// Mitsubishi GX Works2 project: KhanhHungTap2FX3U   PLC: FX3U/FX3UC

// global labels: Global1
VAR_GLOBAL
  XXLimitN AT M8344 : BOOL;
  XXLimitP AT M8343 : BOOL;
  XXBusy AT M8340 : BOOL;
  XXInterruptInverse AT M8347 : BOOL;
  XXPos AT D8340 : DINT;
  XXAccelTime AT D8348 : INT;
  XXDecelTime AT D8349 : INT;
  XXPosView AT D0 : DINT;
  XXTarPos AT D2 : DINT;
  XXFeed AT D4 : DINT;
  XXPPR AT D6 : DINT;
  XXTarR AT M0 : BOOL;
  XXTarRSkip AT D8 : INT;
  XXOn AT M1 : BOOL;
  XXRun AT M2 : BOOL;
  XXDirection AT M3 : BOOL;
  XXMinI AT X000 : BOOL;
  XXReadyI AT X004 : BOOL;
  XXPulseO AT Y000 : BOOL;
  XXDirectionO AT Y004 : BOOL;
  XXOnO AT Y003 : BOOL;
  YYLimitN AT M8354 : BOOL;
  YYLimitP AT M8353 : BOOL;
  YYBusy AT M8350 : BOOL;
  YYInterruptInverse AT M8357 : BOOL;
  YYPos AT D8350 : DINT;
  YYAccelTime AT D8358 : INT;
  YYDecelTime AT D8359 : INT;
  YYPosView AT D9 : DINT;
  YYTarPos AT D11 : DINT;
  YYFeed AT D13 : DINT;
  YYPPM AT D15 : DINT;
  YYTarR AT M4 : BOOL;
  YYTarRSkip AT D17 : INT;
  YYOn AT M5 : BOOL;
  YYRun AT M6 : BOOL;
  YYDirection AT M7 : BOOL;
  YYMinI AT X001 : BOOL;
  YYReadyI AT X005 : BOOL;
  YYPulseO AT Y001 : BOOL;
  YYDirectionO AT Y005 : BOOL;
  YYOnO AT Y007 : BOOL;
  ZZLimitN AT M8364 : BOOL;
  ZZLimitP AT M8363 : BOOL;
  ZZBusy AT M8360 : BOOL;
  ZZInterruptInverse AT M8367 : BOOL;
  ZZPos AT D8360 : DINT;
  ZZAccelTime AT D8368 : INT;
  ZZDecelTime AT D8369 : INT;
  ZZPosView AT D18 : DINT;
  ZZTarPos AT D20 : DINT;
  ZZFeed AT D22 : DINT;
  ZZPPR AT D24 : DINT;
  ZZTarR AT M8 : BOOL;
  ZZTarRSkip AT D26 : INT;
  ZZRun AT M9 : BOOL;
  ZZDirection AT M10 : BOOL;
  ZZReadyI AT X006 : BOOL;
  ZZPulseO AT Y002 : BOOL;
  ZZDirectionO AT Y006 : BOOL;
  ZZOnO AT Y010 : BOOL;
  Run AT M11 : BOOL;
  RunI AT X002 : BOOL;
  RunStop AT M12 : BOOL;
  RunStopI AT X003 : BOOL;
  RunState AT D27 : INT;
  RunStateNext AT M13 : BOOL;
  AxisSpinState AT D28 : INT;
  AxisSpinStateNext AT M14 : BOOL;
  AxisTapState AT D29 : INT;
  AxisTapStateNext AT M15 : BOOL;
  FoilExtractState AT D30 : INT;
  FoilExtractStateNext AT M16 : BOOL;
  FoilClampState AT D31 : INT;
  FoilClampStateNext AT M17 : BOOL;
  FoilSupplyState AT D32 : INT;
  FoilSupplyStateNext AT M18 : BOOL;
  FoilExtractDropN AT M19 : BOOL;
  FoilExtractDropNTimer AT TC0 : BOOL;
  FoilExtractDropNTimerDelay AT D33 : INT;
  FoilExtractDropP AT M20 : BOOL;
  FoilExtractDropPTimer AT TC1 : BOOL;
  FoilExtractDropPTimerDelay AT D34 : INT;
  FoilExtractDrop AT M21 : BOOL;
  FoilExtractDropO AT Y011 : BOOL;
  FoilExtractPushN AT M22 : BOOL;
  FoilExtractPushNTimer AT TC2 : BOOL;
  FoilExtractPushNTimerDelay AT D35 : INT;
  FoilExtractPushP AT M23 : BOOL;
  FoilExtractPushPTimer AT TC3 : BOOL;
  FoilExtractPushPTimerDelay AT D36 : INT;
  FoilExtractPush AT M24 : BOOL;
  FoilExtractPushO AT Y012 : BOOL;
  FoilClampN AT M25 : BOOL;
  FoilClampNTimer AT TC4 : BOOL;
  FoilClampNTimerDelay AT D37 : INT;
  FoilClampP AT M26 : BOOL;
  FoilClampPTimer AT TC5 : BOOL;
  FoilClampPTimerDelay AT D38 : INT;
  FoilClampNI AT X007 : BOOL;
  FoilClampPI AT X010 : BOOL;
  FoilClamp AT M27 : BOOL;
  FoilClampO AT Y013 : BOOL;
  FoilSupplyN AT M28 : BOOL;
  FoilSupplyNTimer AT TC6 : BOOL;
  FoilSupplyNTimerDelay AT D39 : INT;
  FoilSupplyP AT M29 : BOOL;
  FoilSupplyPTimer AT TC7 : BOOL;
  FoilSupplyPTimerDelay AT D40 : INT;
  FoilSupply AT M30 : BOOL;
  FoilSupplyO AT Y014 : BOOL;
  WorkFeedSpin AT D41 : DINT;
  WorkFeedTapSpin AT D43 : DINT;
  WorkFeedTapSpinUp AT D45 : DINT;
  FoilFull AT M31 : BOOL;
  FoilFullI AT X011 : BOOL;
  FoilFullTimer AT TC8 : BOOL;
  SpinArray AT D47 : ARRAY [0..7] OF DINT;
  SpinArrayIndex AT D63 : INT;
  SpinTest AT M32 : BOOL;
  SpinTestTimer AT TC9 : BOOL;
  SpinTestTimerDelay AT D64 : INT;
  SettingTapPitchI AT X012 : BOOL;
  SettingTapPitch AT D65 : DINT;
  SettingTapSpinSpeed1I AT X013 : BOOL;
  SettingTapSpinSpeed2I AT X014 : BOOL;
  SettingTapTravelBegin AT D67 : DINT;
  SettingFoilSupplyI AT X015 : BOOL;
  AirReady AT M33 : BOOL;
  AirReadyI AT X016 : BOOL;
  TapMoveToTravelBegin AT M34 : BOOL;
  TapCount AT D69 : DINT;
  TapCountAtSupplyEnd AT D71 : DINT;
  StopTap AT M35 : BOOL;
  StopTapTimer AT TC10 : BOOL;
  StopClamp AT M36 : BOOL;
  StopClampPLS AT M37 : BOOL;
  StopClampTimer AT TC11 : BOOL;
  FoilSupplyPTimeoutTimer AT TC12 : BOOL;
  FoilSupplyPTimeoutTimerDelay AT D73 : INT;
  XXOff AT M38 : BOOL;
  XXOffTimer AT TC13 : BOOL;
END_VAR

// task Task_01 (event TRUE, interval 0, priority 31): POU_01

PROGRAM POU_01
VAR
  fTmp : BOOL;
  fSpace : DINT;
  fCount : INT;
END_VAR
SET(M8002, M8336);
MOV(M8002, HFFF0, D8336);
RST(M8002, XXInterruptInverse);
RST(M8002, XXOn);
RST(M8002, YYOn);
MOV(M8002, 50, XXAccelTime);
MOV(M8002, 50, XXDecelTime);
MOV(M8002, 150, YYAccelTime);
MOV(M8002, 150, YYDecelTime);
RST(M8002, FoilExtractDrop);
RST(M8002, FoilExtractPush);
RST(M8002, SpinTest);
(*x axis: index spin*)
DMOV(M8002, 131_072, XXPPR);
MOV(M8002, 8, fCount);
DMOV(M8002, XXPPR / INT_TO_DINT(fCount), fSpace);
DMOV(M8002, fSpace * 0, SpinArray[0]);
DMOV(M8002, fSpace * 1, SpinArray[1]);
DMOV(M8002, fSpace * 2, SpinArray[2]);
DMOV(M8002, fSpace * 3, SpinArray[3]);
DMOV(M8002, fSpace * 4, SpinArray[4]);
DMOV(M8002, fSpace * 5, SpinArray[5]);
DMOV(M8002, fSpace * 6, SpinArray[6]);
DMOV(M8002, fSpace * 7, SpinArray[7]);
DMOV(M8002, 98_304, WorkFeedSpin);
(*y axis: tap travel*)
DMOV(M8002, 1_000, YYPPM);
RST(M8002, TapCount);
(*z axis: tap spin*)
DMOV(M8002, YYPPM, ZZPPR);
DMOV(M8002, (ZZPPR * 2_800) / 60, WorkFeedTapSpinUp);
(*it easier to calculate if YYPPM = ZZPPR*)
(*|||||||||||||||*)
(*|||||||||||||||*)
SET(Run AND RunState = 0 AND AirReady, fTmp);
RST(fTmp, Run);
SET(fTmp, XXOn);
SET(fTmp, YYOn);
SET(fTmp, TapMoveToTravelBegin);
RST(fTmp, StopClamp);
MOV(fTmp, 1, RunState);
RST(fTmp, fTmp);
SET(RunStop, fTmp);
RST(fTmp, Run);
RST(fTmp, RunStop);
ZRST(fTmp, RunState, FoilSupplyState);
RST(fTmp, XXRun);
RST(fTmp, XXOn);
RST(fTmp, YYRun);
RST(fTmp, ZZRun);
SET(fTmp AND YYOn, StopTap);
RST(fTmp, FoilExtractDrop);
RST(fTmp, FoilExtractPush);
RST(fTmp, FoilClamp);
RST(fTmp, FoilSupply);
RST(fTmp, fTmp);
OUT_T(StopTap, StopTapTimer, 5);
RST(StopTapTimer, YYOn);
RST(StopTapTimer, StopTap);

(*|||||||||||||||*)
(*|||||||||||||||*)
INC(RunStateNext, RunState);
INC(AxisSpinStateNext, AxisSpinState);
INC(AxisTapStateNext, AxisTapState);
INC(FoilExtractStateNext, FoilExtractState);
INC(FoilClampStateNext, FoilClampState);
INC(FoilSupplyStateNext, FoilSupplyState);
ZRST(M8000, RunStateNext, FoilSupplyStateNext);
DECO(M8000, RunState, 6, M100);
DECO(M8000, AxisSpinState, 6, M200); DECO(M8000, AxisSpinState, 6, M1200); ZRST(NOT XXTarR OR NOT XXReadyI, M1200, M1263);
DECO(M8000, AxisTapState, 6, M300); DECO(M8000, AxisTapState, 6, M1300); ZRST(NOT YYTarR OR NOT YYReadyI OR NOT ZZTarR OR NOT ZZReadyI, M1300, M1363);
DECO(M8000, FoilExtractState, 6, M400);
DECO(M8000, FoilClampState, 6, M500);
DECO(M8000, FoilSupplyState, 6, M600);
(*|||||||||||||||*)

(*|||||||||||||||*)
(*origin tap, extract, clamp, supply*)
MOV(M101, 1, AxisTapState);
MOV(M101, 1, FoilExtractState);
MOV(M101, 1, FoilClampState);
MOV(M101, 1, FoilSupplyState);
DMOV(M101, TapCount - 4, TapCountAtSupplyEnd);
SET(M101, RunStateNext);
(*origin spin*)
MOV(M102 AND M1320, 1, AxisSpinState);
SET(M102 AND M1320, RunStateNext);
(*ready done, foil supply ready, run command -> cycle start*)
SET(M103 AND M1220 AND M1320 AND M420 AND M520 AND Run, RunStateNext);
(*cycle start*)
SET(M104 AND M1220 AND M1320 AND M420 AND M520, RunStateNext);
(*clamp on*)
MOV(M105, 11, FoilClampState);
SET(M105, XXOff);
SET(M105, RunStateNext);
(*clamp on done -> tap, extract*)
SET(M106 AND M515, fTmp);
MOV(fTmp, 11, AxisTapState);
MOV(fTmp, 11, FoilExtractState);
SET(fTmp, RunStateNext);
RST(fTmp, fTmp);
(*tap done -> add tap count, clamp off*)
SET(M107 AND M1320, fTmp);
DINC(fTmp, TapCount);
MOV(fTmp, 16, FoilClampState);
SET(fTmp, RunStateNext);
RST(fTmp, fTmp);
(*clamp off done, extract done -> next hole*)
SET(M108 AND M520 AND M420, fTmp);
MOV(fTmp, 11, AxisSpinState);
SET(fTmp, XXOn);
SET(fTmp, RunStateNext);
RST(fTmp, fTmp);
(*next hole done -> next*)
SET(M109 AND M1220, RunStateNext);
(*return cycle start*)
MOV(M110, 4, RunState);
(*|||||||||||||||*)
(*foil full -> record*)
DMOV(FoilFull, TapCount, TapCountAtSupplyEnd);
(*check*)
SET((TapCount - TapCountAtSupplyEnd) >= 4, fTmp);
RST(NOT SettingFoilSupplyI, fTmp);
MOV(NOT FoilFull AND M620 AND fTmp, 11, FoilSupplyState);
RST(fTmp, fTmp);
(*|||||||||||||||*)

(*|||||||||||||||*)
(*/////get origin spin*)
(*dvit(EN, offset, frequency)*)
DDVIT(M201, 16_384, 32_768, XXPulseO, XXDirection);
SET(M201 AND M8029, AxisSpinStateNext);
RST(M201 AND M8029, M201);
(*reset index and position*)
RST(M1202, SpinArrayIndex);
DMOV(M1202, -fSpace, XXPos);
MOV(M1202, 20, AxisSpinState);
(*reset index and position*)
RST(M1206, SpinArrayIndex);
DMOV(M1206, -fSpace, XXPos);
MOV(M1206, 12, AxisSpinState);
(*/////main sequence*)
(*re get origin or next*)
SET(M1211 AND SpinArrayIndex >= fCount, fTmp);
MOV(M1211 AND fTmp, fCount, AxisSpinState);
SET(M1211 AND NOT fTmp, AxisSpinStateNext);
RST(fTmp, fTmp);
(*move to hole*)
DMOV(M1212, SpinArray[SpinArrayIndex], XXTarPos);
DMOV(M1212, WorkFeedSpin, XXFeed);
INC(M1212, SpinArrayIndex);
SET(M1212, XXRun);
SET(M1212, AxisSpinStateNext);
(*target reach*)
RST(M1213, XXRun);
SET(M1213, AxisSpinStateNext);
(*move to hole done, end*)
SET(M1214, fTmp);
MOV(fTmp, 20, AxisSpinState);
RST(fTmp, fTmp);
(*test*)
OUT_T(M1220 AND SpinTest, SpinTestTimer, SpinTestTimerDelay);
MOV(SpinTestTimer, 11, AxisSpinState);
(*|||||||||||||||*)


(*|||||||||||||||*)
(*/////get origin tap*)
(*at min, jump to move down*)
SET(M301 AND YYMinI, fTmp);
MOV(fTmp, 2, AxisTapState);
RST(fTmp, fTmp);
(*not at min, move up*)
SET(M1301 AND NOT YYMinI, fTmp);
RST(fTmp, YYPos); RST(fTmp, ZZPos);
DMOV(fTmp, -100_000, YYTarPos); DMOV(fTmp, YYTarPos * ZZPPR / SettingTapPitch, ZZTarPos);
DMOV(fTmp, 5_000, YYFeed); DMOV(fTmp, YYFeed * ZZPPR / SettingTapPitch, ZZFeed);
SET(fTmp, YYRun); SET(fTmp, ZZRun);
SET(fTmp, AxisTapStateNext);
RST(fTmp, fTmp);
(*move up hit limit -> reset*)
SET(M302 AND NOT YYBusy, fTmp);
RST(fTmp, YYRun); RST(fTmp, ZZRun);
RST(fTmp, YYPos); RST(fTmp, ZZPos);
SET(fTmp, AxisTapStateNext);
RST(fTmp, fTmp);
(*move down*)
SET(M1303, fTmp);
DMOV(fTmp, 5_000, YYTarPos);
DMOV(fTmp, 1_000, YYFeed);
SET(fTmp, YYRun);
SET(fTmp, AxisTapStateNext);
RST(fTmp, fTmp);
(*move down out min, stop*)
SET(M304 AND NOT YYMinI, fTmp);
RST(fTmp, YYRun);
SET(fTmp, AxisTapStateNext);
RST(fTmp, fTmp);
(*stop done, move down x mm*)
SET(M1305, fTmp);
DMOV(fTmp, YYPos + 5_000, YYTarPos);
DMOV(fTmp, 1_000, YYFeed);
SET(fTmp, YYRun);
SET(fTmp, AxisTapStateNext);
RST(fTmp, fTmp);
(*move down x mm done -> reset, move to begin or end*)
SET(M1306, fTmp);
RST(fTmp, YYPos); RST(fTmp, ZZPos);
MOV(fTmp AND TapMoveToTravelBegin, 7, AxisTapState);
MOV(fTmp AND NOT TapMoveToTravelBegin, 8, AxisTapState);
RST(fTmp, fTmp);
(*move to begin*)
DMOV(M1307, SettingTapTravelBegin, YYTarPos);
DMOV(M1307, 5_000, YYFeed);
SET(M1307, YYRun);
SET(M1307, AxisTapStateNext);
(*ready*)
MOV(M1308, 20, AxisTapState);
(*/////main sequence*)
(*move down*)
SET(M1311, fTmp);
DMOV(fTmp, 35_000, YYTarPos); RST(fTmp, ZZPos); DMOV(fTmp, (YYTarPos - YYPos) * ZZPPR / SettingTapPitch, ZZTarPos);
DMOV(fTmp, WorkFeedTapSpin, ZZFeed); DMOV(fTmp, ZZFeed * SettingTapPitch / ZZPPR, YYFeed);
SET(fTmp, YYRun); SET(fTmp, ZZRun);
SET(fTmp, AxisTapStateNext); RST(fTmp, fTmp);
(*target reach or touch max, reset*)
SET(M1312 OR (M312 AND NOT YYBusy), fTmp);
RST(fTmp, YYRun); RST(fTmp, ZZRun);
SET(fTmp, AxisTapStateNext); RST(fTmp, fTmp);
(*move down done, move up*)
SET(M1313, fTmp);
DMOV(fTmp, SettingTapTravelBegin, YYTarPos); RST(fTmp, ZZPos); DMOV(fTmp, (YYTarPos - YYPos) * ZZPPR / SettingTapPitch, ZZTarPos);
DMOV(fTmp, WorkFeedTapSpinUp, ZZFeed); DMOV(fTmp, ZZFeed * SettingTapPitch / ZZPPR, YYFeed);
SET(fTmp, YYRun); SET(fTmp, ZZRun);
SET(fTmp, AxisTapStateNext); RST(fTmp, fTmp);
(*move up done, return wait tap hit*)
SET(M1314, fTmp);
MOV(fTmp, 20, AxisTapState); RST(fTmp, fTmp);
(*|||||||||||||||*)

(*|||||||||||||||*)
(*/////get origin foil extract*)
(*drop back, push back*)
RST(M401, FoilExtractDrop);
RST(M401, FoilExtractPush);
SET(M401, FoilExtractStateNext);
(*drop back done, push forward done -> next*)
SET(M402 AND FoilExtractDropN AND FoilExtractPushN, FoilExtractStateNext);
(*end*)
MOV(M403, 20, FoilExtractState);
(*/////main sequence*)
(*drop forward*)
SET(M411, FoilExtractDrop);
SET(M411, FoilExtractStateNext);
(*drop forward done -> drop back*)
RST(M412 AND FoilExtractDropP, FoilExtractDrop);
SET(M412 AND FoilExtractDropP, FoilExtractStateNext);
(*drop back done -> push forward*)
SET(M413 AND FoilExtractDropN, FoilExtractPush);
SET(M413 AND FoilExtractDropN, FoilExtractStateNext);
(*push forward done -> push back*)
RST(M414 AND FoilExtractPushP, FoilExtractPush);
SET(M414 AND FoilExtractPushP, FoilExtractStateNext);
(*push back done -> end*)
MOV(M415 AND FoilExtractPushN, 20, FoilExtractState);
(*|||||||||||||||*)

(*|||||||||||||||*)
(*/////get origin foil clamp*)

(*back*)
RST(M501, FoilClamp);
SET(M501, FoilClampStateNext);
(*back done -> next*)
SET(M502 AND FoilClampN, FoilClampStateNext);
(*end*)
MOV(M503, 20, FoilClampState);
(*/////clamp on*)
(*forward*)
SET(M511, FoilClamp);
SET(M511, FoilClampStateNext);
(*forward done -> done*)
MOV(M512 AND FoilClampP, 15, FoilClampState);
(*/////clamp off*)
(*back*)
RST(M516, FoilClamp);
SET(M516, FoilClampStateNext);
(*back done -> done*)
MOV(M517 AND FoilClampN, 20, FoilClampState);
(*|||||||||||||||*)

(*|||||||||||||||*)
(*/////get origin foil supply*)
(*down*)
RST(M601, FoilSupply);
SET(M601, FoilSupplyStateNext);
(*down done -> next*)
SET(M602 AND FoilSupplyN, FoilSupplyStateNext);
(*end*)
MOV(M603, 20, FoilSupplyState);
(*/////supply sequence*)
(*up*)
SET(M611, FoilSupply);
SET(M611, FoilSupplyStateNext);
(*up done -> down*)
RST(M612 AND FoilSupplyP, FoilSupply);
SET(M612 AND FoilSupplyP, FoilSupplyStateNext);
(*down done -> end*)
MOV(M613 AND FoilSupplyN, 20, FoilSupplyState);
(*|||||||||||||||*)

(*|||||||||||||||*)
(*XX*)
RST(XXRun AND XXTarPos = XXPos, XXRun);
DDRVA(XXRun, XXTarPos, XXFeed, XXPulseO, XXDirection);
RST(M8029, XXRun);
OUT(XXDirection, XXDirectionO);
INC(NOT XXRun AND NOT XXBusy AND XXTarRSkip < 5, XXTarRSkip);
RST(XXRun, XXTarRSkip);
OUT(XXTarRSkip >= 5, XXTarR);
(*|||||||||||||||*)
(*YY*)
RST(YYRun AND YYTarPos = YYPos, YYRun);
DDRVA(YYRun, YYTarPos, YYFeed, YYPulseO, YYDirection);
RST(M8029, YYRun);
OUT(NOT YYDirection, YYDirectionO);
INC(NOT YYRun AND NOT YYBusy AND YYTarRSkip < 5, YYTarRSkip);
RST(YYRun, YYTarRSkip);
OUT(YYTarRSkip >= 5, YYTarR);
(**)
OUT(YYMinI, YYLimitN);
(*|||||||||||||||*)
(*ZZ*)
RST(ZZRun AND ZZTarPos = ZZPos, ZZRun);
DDRVA(ZZRun, ZZTarPos, ZZFeed, ZZPulseO, ZZDirection);
RST(M8029, ZZRun);
OUT(NOT ZZDirection, ZZDirectionO);
INC(NOT ZZRun AND NOT ZZBusy AND ZZTarRSkip < 5, ZZTarRSkip);
RST(ZZRun, ZZTarRSkip);
OUT(ZZTarRSkip >= 5, ZZTarR);
(**)
OUT(YYMinI, ZZLimitN);
(*|||||||||||||||*)

(*|||||||||||||||*)
PLS(RunI, Run); SET(Run, Run);
PLF(RunStopI, RunStop); SET(RunStop, RunStop);
OUT_T(NOT RunStopI AND NOT StopClamp, StopClampTimer, 20); SET(StopClampTimer, StopClamp);
RST(StopClamp, RunStop);
SET(StopClamp, FoilClamp);
SET(StopClamp AND FoilClampP, fTmp);
SET(fTmp, YYOn);
MOV(fTmp, 1, AxisTapState);
RST(fTmp, StopClamp);
RST(fTmp, TapMoveToTravelBegin);
RST(fTmp, fTmp);
(**)
MOV(M8002, 2, FoilExtractDropNTimerDelay);
OUT_T(NOT FoilExtractDrop, FoilExtractDropNTimer, FoilExtractDropNTimerDelay); SET(FoilExtractDropNTimer, FoilExtractDropN); RST(FoilExtractDropNTimer, FoilExtractDropP);
MOV(M8002, 2, FoilExtractDropPTimerDelay);
OUT_T(FoilExtractDrop, FoilExtractDropPTimer, FoilExtractDropPTimerDelay); SET(FoilExtractDropPTimer, FoilExtractDropP); RST(FoilExtractDropPTimer, FoilExtractDropN);
MOV(M8002, 2, FoilExtractPushNTimerDelay);
OUT_T(NOT FoilExtractPush, FoilExtractPushNTimer, FoilExtractPushNTimerDelay); SET(FoilExtractPushNTimer, FoilExtractPushN); RST(FoilExtractPushNTimer, FoilExtractPushP);
MOV(M8002, 2, FoilExtractPushPTimerDelay);
OUT_T(FoilExtractPush, FoilExtractPushPTimer, FoilExtractPushPTimerDelay); SET(FoilExtractPushPTimer, FoilExtractPushP); RST(FoilExtractPushPTimer, FoilExtractPushN);
(**)
MOV(M8002, 1, FoilClampNTimerDelay);
OUT_T(NOT FoilClamp AND FoilClampNI, FoilClampNTimer, FoilClampNTimerDelay); SET(FoilClampNTimer, FoilClampN); RST(FoilClampNTimer, FoilClampP);
MOV(M8002, 1, FoilClampPTimerDelay);
OUT_T(FoilClamp AND FoilClampPI, FoilClampPTimer, FoilClampPTimerDelay); SET(FoilClampPTimer, FoilClampP); RST(FoilClampPTimer, FoilClampN);
(**)
MOV(M8002, 10, FoilSupplyNTimerDelay);
OUT_T(NOT FoilSupply, FoilSupplyNTimer, FoilSupplyNTimerDelay); SET(FoilSupplyNTimer, FoilSupplyN); RST(FoilSupplyNTimer, FoilSupplyP);
MOV(M8002, 18, FoilSupplyPTimerDelay);
OUT_T(FoilSupply, FoilSupplyPTimer, FoilSupplyPTimerDelay); SET(FoilSupplyPTimer, FoilSupplyP); RST(FoilSupplyPTimer, FoilSupplyN);
MOV(M8002, 40, FoilSupplyPTimeoutTimerDelay);
OUT_T(FoilSupply, FoilSupplyPTimeoutTimer, FoilSupplyPTimeoutTimerDelay); SET(FoilSupplyPTimeoutTimer, FoilSupplyP); RST(FoilSupplyPTimeoutTimer, FoilSupplyN);
(**)
OUT_T(FoilFullI, FoilFullTimer, 8); OUT(FoilFullTimer, FoilFull);
(*setting feed*)
DMOV(SettingTapSpinSpeed1I, (ZZPPR * 1_200) / 60, WorkFeedTapSpin);
DMOV(NOT (SettingTapSpinSpeed1I OR SettingTapSpinSpeed2I), (ZZPPR * 1_600) / 60, WorkFeedTapSpin);
DMOV(SettingTapSpinSpeed2I, (ZZPPR * 2_000) / 60, WorkFeedTapSpin);
(*setting pitch*)
DMOV(SettingTapPitchI, 1_000, SettingTapPitch);
DMOV(NOT SettingTapPitchI, 1_270, SettingTapPitch);
(*setting travel*)
DMOV(M8002, 5_000, SettingTapTravelBegin);
(**)
OUT(AirReadyI, AirReady);
(*|||||||||||||||*)
OUT(XXOn, XXOnO);
OUT(YYOn, YYOnO); OUT(YYOn, ZZOnO);
OUT(FoilExtractDrop, FoilExtractDropO);
OUT(FoilExtractPush, FoilExtractPushO);
OUT(FoilClamp, FoilClampO);
OUT(FoilSupply, FoilSupplyO);
OUT_T(XXOff, XXOffTimer, 2); RST(XXOffTimer, XXOn); RST(XXOffTimer, XXOff);
(*|||||||||||||||*)
END_PROGRAM
